(* Logix 5000 project; controller test vendor 1 type 14 code 65 rev 20.19; software revision 20.04 *)

TASK MainTask (continuous, watchdog 500 ms) : HallwaySensor, MapInputs, DoorSensor

MODULES
   Controller : vendor 1 type 14 code 65 (CompactLogixL35Controller 0, rev 20.19)
      LocalENB : 1769-L35E Ethernet Port (CompactLogixL35Ethernet 1, rev 20.11)
      Local : CompactBus (CompactVirtualAdapter 3, rev 20.11)
         digital : vendor 1 type 7 code 66 (Compact 2, rev 1.1, Output RPI 20 ms)
         Analog : vendor 1 type 10 code 33 (Compact 1, rev 1.1, Output RPI 80 ms)
END_MODULES

VAR_GLOBAL   (* controller tags *)
   ak47_obj : BOOL;
   door_snsr_status : ALIAS FOR Local:2:I.Data.0;
   hallway_snsr_status : ALIAS FOR Local:2:I.Data.1;
END_VAR

PROGRAM AK47Detector
END_PROGRAM

PROGRAM DoorSensor
VAR
   door_snsr_in : ALIAS FOR Local:2:I.Data.0;   // From front door sensor (yellow wire)
   door_snsr_out : ALIAS FOR Local:2:O.Data.0;
END_VAR

ROUTINE Ab_Main   (* ladder *)
// Routine for the front door sensor
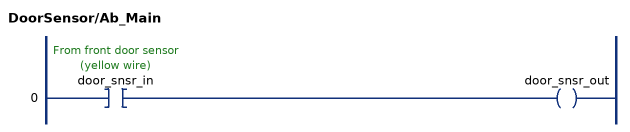
   0 (stored rung type 13): XIC(door_snsr_in)OTE(door_snsr_out);
END_ROUTINE
END_PROGRAM

PROGRAM Faults
END_PROGRAM

PROGRAM HallwaySensor   (* main routine Aa_Main *)
VAR
   hallway_snsr_in : ALIAS FOR Local:2:I.Data.1;   // The white wire input from the Photo Eye sensor in the hallway.
END_VAR

ROUTINE Aa_Main   (* ladder *)
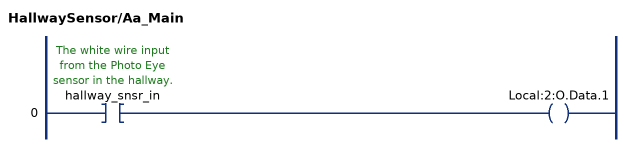
   0 (stored rung type 13): XIC(hallway_snsr_in)OTE(Local:2:O.Data.1);
END_ROUTINE
END_PROGRAM

PROGRAM MapInputs
VAR
   light : ALIAS FOR Local:2:O.Data.0;
   start_switch : ALIAS FOR Local:2:I.Data.0;   // test switch
END_VAR

ROUTINE MainRoutine   (* ladder *)
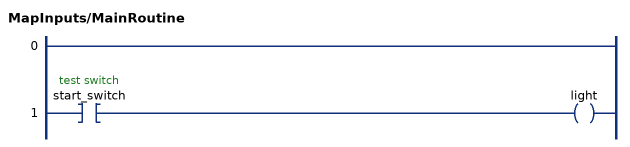
   0 (stored rung type 13): ;
   1 (stored rung type 1): XIC(start_switch)OTE(light);
END_ROUTINE
END_PROGRAM
